(* IEC 61131-3 sources: plc_generation_empirical_study/datasets/task_bank_c06_reverse_bounded_runtime_v0_3/tasks/C06_V19_lean_composite, 2 files *)

(* ---- interface.st ---- *)
FUNCTION_BLOCK C06_V19_lean_composite
VAR_INPUT
    A_AutoMode : BOOL;
    A_AutoDemand : BOOL;
    A_ManualDemand : BOOL;
    A_SafetyOK : BOOL;
    A_Inhibit : BOOL;
    B_AddItem : BOOL;
    B_RemoveItem : BOOL;
    B_Reset : BOOL;
    B_Capacity : INT;
    SubsystemBEnable : BOOL;
    CrossReset : BOOL;
END_VAR
VAR_OUTPUT
    A_Command : BOOL;
    A_Blocked : BOOL;
    B_Count : INT;
    B_Empty : BOOL;
    B_Full : BOOL;
    B_Conflict : BOOL;
    CrossReady : BOOL;
    CrossBlocked : BOOL;
END_VAR
END_FUNCTION_BLOCK

(* ---- reference.st ---- *)
FUNCTION_BLOCK C06_V19_lean_composite
VAR_INPUT
    A_AutoMode : BOOL;
    A_AutoDemand : BOOL;
    A_ManualDemand : BOOL;
    A_SafetyOK : BOOL;
    A_Inhibit : BOOL;
    B_AddItem : BOOL;
    B_RemoveItem : BOOL;
    B_Reset : BOOL;
    B_Capacity : INT;
    SubsystemBEnable : BOOL;
    CrossReset : BOOL;
END_VAR
VAR_OUTPUT
    A_Command : BOOL;
    A_Blocked : BOOL;
    B_Count : INT;
    B_Empty : BOOL;
    B_Full : BOOL;
    B_Conflict : BOOL;
    CrossReady : BOOL;
    CrossBlocked : BOOL;
END_VAR
VAR
    B_PrevAdd : BOOL := FALSE;
    B_PrevRemove : BOOL := FALSE;
END_VAR

A_Command := ((A_AutoMode AND A_AutoDemand) OR ((NOT A_AutoMode) AND A_ManualDemand))
           AND A_SafetyOK AND (NOT A_Inhibit);
A_Blocked := ((A_AutoMode AND A_AutoDemand) OR ((NOT A_AutoMode) AND A_ManualDemand))
           AND ((NOT A_SafetyOK) OR A_Inhibit);

IF CrossReset THEN
    CrossReady := FALSE;
ELSIF A_Command THEN
    CrossReady := TRUE;
END_IF;
CrossBlocked := SubsystemBEnable AND (NOT CrossReady);

IF SubsystemBEnable AND CrossReady THEN
    B_Conflict := FALSE;
    IF B_Reset THEN
        B_Count := 0;
    ELSIF B_AddItem AND (NOT B_PrevAdd) AND B_RemoveItem AND (NOT B_PrevRemove) THEN
        B_Conflict := TRUE;
    ELSIF B_AddItem AND (NOT B_PrevAdd) AND (B_Count < B_Capacity) THEN
        B_Count := B_Count + 1;
    ELSIF B_RemoveItem AND (NOT B_PrevRemove) AND (B_Count > 0) THEN
        B_Count := B_Count - 1;
    END_IF;
    B_Empty := B_Count = 0;
    B_Full := B_Count >= B_Capacity;
    B_PrevAdd := B_AddItem;
    B_PrevRemove := B_RemoveItem;
ELSE
    B_Count := 0;
    B_Empty := FALSE;
    B_Full := FALSE;
    B_Conflict := FALSE;
END_IF;

END_FUNCTION_BLOCK
